(* CODESYS project Mini_Project.project

Project tree, tasks and I/O mapping:
  Device : CECC-LK, Festo AG & Co. KG, order no. 574418, version 3.5.4.0
    application Application
      libraries: Standard, * (System); Solution Center Library, 3.5.8.0 (Festo Didactic SE - Customer Solution Center); CAA CiA 405, 3.5.3.0 (CAA Technical Workgroup)
      task MainTask (cyclic, interval t#20ms, priority 20) calls PLC_PRG
      program PLC_PRG [ST]
      function block TCP_Conn [ST]
      function block RFID_Read [ST]
      function block SPLIT_String [ST]
      function formatMsg [ST]
    Onboard : CECC 14I/8O, Festo AG & Co. KG, version 3.4.5.5
        unmapped channels: Onboard Input, Onboard Output
      Digital Inputs
          unmapped channels: Onboard Input
      Digital Outputs
          unmapped channels: Onboard Output
    CANbus : CANbus, 3S - Smart Software Solutions GmbH, version 3.5.7.0
        settings: Baudrate = 1000
      CANopen_Manager : CANopen_Manager, 3S - Smart Software Solutions GmbH, version 3.5.10.0
          settings: ConfigVersion = 50659584
        BL20_GWBR_CANOPEN : BL20-GWBR-CANOPEN, TURCK, order no. 6827167, version Revision=16#00040017, FileVersion=4.23
            settings: General Options.Reset Node = FALSE; NODEIDSAVED = 2; SDO Timeout = 1000000; PDO_Autoconfig = TRUE; EXPERTSETTINGS = True; Emergency-General Parameters.Emergency COBID = 16#00000082; Settings.COBID = 16#00000202; Settings.Transmission Type = 16#FF; Settings.available PDO-Parameter.Inhibit Time available = FALSE; Settings.available PDO-Parameter.Event Timer available = FALSE; Settings.Inhibit Time = 0; Settings.Event Timer = 0; Generic COBID = '$NODEID+16#0200'; Settings.COBID = 16#00000302; Settings.Transmission Type = 16#FF; Settings.available PDO-Parameter.Inhibit Time available = FALSE; Settings.available PDO-Parameter.Event Timer available = FALSE; Settings.Inhibit Time = 0; Settings.Event Timer = 0; Generic COBID = '$NODEID+16#0300'; Settings.COBID = 16#00000182; Settings.Transmission Type = 16#FF; Settings.available PDO-Parameter.Inhibit Time available = TRUE; Settings.available PDO-Parameter.Event Timer available = TRUE; Settings.Inhibit Time = 0; Settings.Event Timer = 0; Generic COBID = '$NODEID+16#0180'; Settings.COBID = 16#00000282; Settings.Transmission Type = 16#FF; Settings.available PDO-Parameter.Inhibit Time available = TRUE; Settings.available PDO-Parameter.Event Timer available = TRUE; Settings.Inhibit Time = 0; Settings.Event Timer = 0; Generic COBID = '$NODEID+16#0280'; Heartbeat-Consuming1.Heartbeat-Time = 300 ms; WriteOutput8Bit : Generic_BL20_4DO.Index = 16#6200; WriteOutput8Bit : Generic_BL20_4DO.Subindex = 16#01; WriteOutput8Bit : Generic_BL20_4DO.ObjectLength = 8; WriteOutput8Bit : Generic_BL20_4DO_2.Index = 16#6200; WriteOutput8Bit : Generic_BL20_4DO_2.Subindex = 16#02;
              WriteOutput8Bit : Generic_BL20_4DO_2.ObjectLength = 8; WriteAnalogueOutput16 : Generic_BL20_2AO.Index = 16#6411; WriteAnalogueOutput16 : Generic_BL20_2AO.Subindex = 16#01; WriteAnalogueOutput16 : Generic_BL20_2AO.ObjectLength = 16; WriteAnalogueOutput16 : Generic_BL20_2AO.Index = 16#6411; WriteAnalogueOutput16 : Generic_BL20_2AO.Subindex = 16#02; WriteAnalogueOutput16 : Generic_BL20_2AO.ObjectLength = 16; ReadInput8Bit : Generic_BL20_4DI.Index = 16#6000; ReadInput8Bit : Generic_BL20_4DI.Subindex = 16#01; ReadInput8Bit : Generic_BL20_4DI.ObjectLength = 8; ReadAnalogueInput16Bit : Generic_BL20_4AI.Index = 16#6401; ReadAnalogueInput16Bit : Generic_BL20_4AI.Subindex = 16#01; ReadAnalogueInput16Bit : Generic_BL20_4AI.ObjectLength = 16; ReadAnalogueInput16Bit : Generic_BL20_4AI.Index = 16#6401; ReadAnalogueInput16Bit : Generic_BL20_4AI.Subindex = 16#02; ReadAnalogueInput16Bit : Generic_BL20_4AI.ObjectLength = 16; ReadAnalogueInput16Bit : Generic_BL20_4AI.Index = 16#6401; ReadAnalogueInput16Bit : Generic_BL20_4AI.Subindex = 16#03; ReadAnalogueInput16Bit : Generic_BL20_4AI.ObjectLength = 16; ReadAnalogueInput16Bit : Generic_BL20_4AI.Index = 16#6401; ReadAnalogueInput16Bit : Generic_BL20_4AI.Subindex = 16#04; ReadAnalogueInput16Bit : Generic_BL20_4AI.ObjectLength = 16; SDO List.Set Guardtime.Index = 16#100C; SDO List.Set Guardtime.Subindex = 16#00; SDO List.Set Guardtime.Value = 16#00000000; SDO List.Set Guardtime.Size = 16; SDO List.Set Guardtime.AbortIfError = FALSE; SDO List.Set Guardtime.JumpToLine = FALSE; SDO List.Set Guardtime.Line = 0; SDO List.Set Lifetime.Index = 16#100D; SDO List.Set Lifetime.Subindex = 16#00; SDO List.Set Lifetime.Value = 16#00000000; SDO List.Set Lifetime.Size = 8; SDO List.Set Lifetime.AbortIfError = FALSE; SDO List.Set Lifetime.JumpToLine = FALSE; SDO List.Set Lifetime.Line = 0; SDO List.Disable Emcy CobID.Index = 16#1014; SDO List.Disable Emcy CobID.Subindex = 16#00; SDO List.Disable Emcy CobID.Value = 16#80000082; SDO List.Disable Emcy CobID.Size = 32;
              SDO List.Disable Emcy CobID.AbortIfError = FALSE; SDO List.Disable Emcy CobID.JumpToLine = FALSE; SDO List.Disable Emcy CobID.Line = 0; SDO List.Set Emcy CobID.Index = 16#1014; SDO List.Set Emcy CobID.Subindex = 16#00; SDO List.Set Emcy CobID.Value = 16#00000082; SDO List.Set Emcy CobID.Size = 32; SDO List.Set Emcy CobID.AbortIfError = FALSE; SDO List.Set Emcy CobID.JumpToLine = FALSE; SDO List.Set Emcy CobID.Line = 0; SDO List.Set Heartbeat Consumer.Index = 16#1016; SDO List.Set Heartbeat Consumer.Subindex = 16#01; SDO List.Set Heartbeat Consumer.Value = 16#007F012C; SDO List.Set Heartbeat Consumer.Size = 32; SDO List.Set Heartbeat Consumer.AbortIfError = FALSE; SDO List.Set Heartbeat Consumer.JumpToLine = FALSE; SDO List.Set Heartbeat Consumer.Line = 0; SDO List.Set Heartbeat Producer.Index = 16#1017; SDO List.Set Heartbeat Producer.Subindex = 16#00; SDO List.Set Heartbeat Producer.Value = 16#00000000; SDO List.Set Heartbeat Producer.Size = 16; SDO List.Set Heartbeat Producer.AbortIfError = FALSE; SDO List.Set Heartbeat Producer.JumpToLine = FALSE; SDO List.Set Heartbeat Producer.Line = 0; SDO List.Disable PDO.Index = 16#1400; SDO List.Disable PDO.Subindex = 16#01; SDO List.Disable PDO.Value = 16#80000202; SDO List.Disable PDO.Size = 32; SDO List.Disable PDO.AbortIfError = FALSE; SDO List.Disable PDO.JumpToLine = FALSE; SDO List.Disable PDO.Line = 0; SDO List.Set transmission type.Index = 16#1400; SDO List.Set transmission type.Subindex = 16#02; SDO List.Set transmission type.Value = 16#FF; SDO List.Set transmission type.Size = 8; SDO List.Set transmission type.AbortIfError = FALSE; SDO List.Set transmission type.JumpToLine = FALSE; SDO List.Set transmission type.Line = 0; SDO List.Clear pdo mapping.Index = 16#1600; SDO List.Clear pdo mapping.Subindex = 16#00;
              SDO List.Clear pdo mapping.Value = 16#0; SDO List.Clear pdo mapping.Size = 8; SDO List.Clear pdo mapping.AbortIfError = FALSE; SDO List.Clear pdo mapping.JumpToLine = FALSE; SDO List.Clear pdo mapping.Line = 0; SDO List.Set Mapping.Index = 16#1600; SDO List.Set Mapping.Subindex = 16#01; SDO List.Set Mapping.Value = 16#62000108; SDO List.Set Mapping.Size = 32; SDO List.Set Mapping.AbortIfError = FALSE; SDO List.Set Mapping.JumpToLine = FALSE; SDO List.Set Mapping.Line = 0; SDO List.Set Mapping.Index = 16#1600; SDO List.Set Mapping.Subindex = 16#02; SDO List.Set Mapping.Value = 16#62000208; SDO List.Set Mapping.Size = 32; SDO List.Set Mapping.AbortIfError = FALSE; SDO List.Set Mapping.JumpToLine = FALSE; SDO List.Set Mapping.Line = 0; SDO List.Set number of mappings.Index = 16#1600; SDO List.Set number of mappings.Subindex = 16#00; SDO List.Set number of mappings.Value = 16#02; SDO List.Set number of mappings.Size = 8; SDO List.Set number of mappings.AbortIfError = FALSE; SDO List.Set number of mappings.JumpToLine = FALSE; SDO List.Set number of mappings.Line = 0; SDO List.Set and enable COB-ID.Index = 16#1400; SDO List.Set and enable COB-ID.Subindex = 16#01; SDO List.Set and enable COB-ID.Value = 16#00000202; SDO List.Set and enable COB-ID.Size = 32; SDO List.Set and enable COB-ID.AbortIfError = FALSE; SDO List.Set and enable COB-ID.JumpToLine = FALSE; SDO List.Set and enable COB-ID.Line = 0; SDO List.Disable PDO.Index = 16#1401; SDO List.Disable PDO.Subindex = 16#01; SDO List.Disable PDO.Value = 16#80000302; SDO List.Disable PDO.Size = 32; SDO List.Disable PDO.AbortIfError = FALSE; SDO List.Disable PDO.JumpToLine = FALSE; SDO List.Disable PDO.Line = 0;
              SDO List.Set transmission type.Index = 16#1401; SDO List.Set transmission type.Subindex = 16#02; SDO List.Set transmission type.Value = 16#FF; SDO List.Set transmission type.Size = 8; SDO List.Set transmission type.AbortIfError = FALSE; SDO List.Set transmission type.JumpToLine = FALSE; SDO List.Set transmission type.Line = 0; SDO List.Clear pdo mapping.Index = 16#1601; SDO List.Clear pdo mapping.Subindex = 16#00; SDO List.Clear pdo mapping.Value = 16#0; SDO List.Clear pdo mapping.Size = 8; SDO List.Clear pdo mapping.AbortIfError = FALSE; SDO List.Clear pdo mapping.JumpToLine = FALSE; SDO List.Clear pdo mapping.Line = 0; SDO List.Set Mapping.Index = 16#1601; SDO List.Set Mapping.Subindex = 16#01; SDO List.Set Mapping.Value = 16#64110110; SDO List.Set Mapping.Size = 32; SDO List.Set Mapping.AbortIfError = FALSE; SDO List.Set Mapping.JumpToLine = FALSE; SDO List.Set Mapping.Line = 0; SDO List.Set Mapping.Index = 16#1601; SDO List.Set Mapping.Subindex = 16#02; SDO List.Set Mapping.Value = 16#64110210; SDO List.Set Mapping.Size = 32; SDO List.Set Mapping.AbortIfError = FALSE; SDO List.Set Mapping.JumpToLine = FALSE; SDO List.Set Mapping.Line = 0; SDO List.Set number of mappings.Index = 16#1601; SDO List.Set number of mappings.Subindex = 16#00; SDO List.Set number of mappings.Value = 16#02; SDO List.Set number of mappings.Size = 8; SDO List.Set number of mappings.AbortIfError = FALSE; SDO List.Set number of mappings.JumpToLine = FALSE; SDO List.Set number of mappings.Line = 0; SDO List.Set and enable COB-ID.Index = 16#1401; SDO List.Set and enable COB-ID.Subindex = 16#01; SDO List.Set and enable COB-ID.Value = 16#00000302; SDO List.Set and enable COB-ID.Size = 32; SDO List.Set and enable COB-ID.AbortIfError = FALSE;
              SDO List.Set and enable COB-ID.JumpToLine = FALSE; SDO List.Set and enable COB-ID.Line = 0; SDO List.Disable PDO.Index = 16#1800; SDO List.Disable PDO.Subindex = 16#01; SDO List.Disable PDO.Value = 16#80000182; SDO List.Disable PDO.Size = 32; SDO List.Disable PDO.AbortIfError = FALSE; SDO List.Disable PDO.JumpToLine = FALSE; SDO List.Disable PDO.Line = 0; SDO List.Set transmission type.Index = 16#1800; SDO List.Set transmission type.Subindex = 16#02; SDO List.Set transmission type.Value = 16#FF; SDO List.Set transmission type.Size = 8; SDO List.Set transmission type.AbortIfError = FALSE; SDO List.Set transmission type.JumpToLine = FALSE; SDO List.Set transmission type.Line = 0; SDO List.Set inhibit time.Index = 16#1800; SDO List.Set inhibit time.Subindex = 16#03; SDO List.Set inhibit time.Value = 16#0000; SDO List.Set inhibit time.Size = 16; SDO List.Set inhibit time.AbortIfError = FALSE; SDO List.Set inhibit time.JumpToLine = FALSE; SDO List.Set inhibit time.Line = 0; SDO List.Set event time.Index = 16#1800; SDO List.Set event time.Subindex = 16#05; SDO List.Set event time.Value = 16#0000; SDO List.Set event time.Size = 16; SDO List.Set event time.AbortIfError = FALSE; SDO List.Set event time.JumpToLine = FALSE; SDO List.Set event time.Line = 0; SDO List.Clear pdo mapping.Index = 16#1A00; SDO List.Clear pdo mapping.Subindex = 16#00; SDO List.Clear pdo mapping.Value = 16#0; SDO List.Clear pdo mapping.Size = 8; SDO List.Clear pdo mapping.AbortIfError = FALSE; SDO List.Clear pdo mapping.JumpToLine = FALSE; SDO List.Clear pdo mapping.Line = 0; SDO List.Set Mapping.Index = 16#1A00; SDO List.Set Mapping.Subindex = 16#01; SDO List.Set Mapping.Value = 16#60000108;
              SDO List.Set Mapping.Size = 32; SDO List.Set Mapping.AbortIfError = FALSE; SDO List.Set Mapping.JumpToLine = FALSE; SDO List.Set Mapping.Line = 0; SDO List.Set number of mappings.Index = 16#1A00; SDO List.Set number of mappings.Subindex = 16#00; SDO List.Set number of mappings.Value = 16#01; SDO List.Set number of mappings.Size = 8; SDO List.Set number of mappings.AbortIfError = FALSE; SDO List.Set number of mappings.JumpToLine = FALSE; SDO List.Set number of mappings.Line = 0; SDO List.Set and enable COB-ID.Index = 16#1800; SDO List.Set and enable COB-ID.Subindex = 16#01; SDO List.Set and enable COB-ID.Value = 16#00000182; SDO List.Set and enable COB-ID.Size = 32; SDO List.Set and enable COB-ID.AbortIfError = FALSE; SDO List.Set and enable COB-ID.JumpToLine = FALSE; SDO List.Set and enable COB-ID.Line = 0; SDO List.Disable PDO.Index = 16#1801; SDO List.Disable PDO.Subindex = 16#01; SDO List.Disable PDO.Value = 16#80000282; SDO List.Disable PDO.Size = 32; SDO List.Disable PDO.AbortIfError = FALSE; SDO List.Disable PDO.JumpToLine = FALSE; SDO List.Disable PDO.Line = 0; SDO List.Set transmission type.Index = 16#1801; SDO List.Set transmission type.Subindex = 16#02; SDO List.Set transmission type.Value = 16#FF; SDO List.Set transmission type.Size = 8; SDO List.Set transmission type.AbortIfError = FALSE; SDO List.Set transmission type.JumpToLine = FALSE; SDO List.Set transmission type.Line = 0; SDO List.Set inhibit time.Index = 16#1801; SDO List.Set inhibit time.Subindex = 16#03; SDO List.Set inhibit time.Value = 16#0000; SDO List.Set inhibit time.Size = 16; SDO List.Set inhibit time.AbortIfError = FALSE; SDO List.Set inhibit time.JumpToLine = FALSE; SDO List.Set inhibit time.Line = 0; SDO List.Set event time.Index = 16#1801;
              SDO List.Set event time.Subindex = 16#05; SDO List.Set event time.Value = 16#0000; SDO List.Set event time.Size = 16; SDO List.Set event time.AbortIfError = FALSE; SDO List.Set event time.JumpToLine = FALSE; SDO List.Set event time.Line = 0; SDO List.Clear pdo mapping.Index = 16#1A01; SDO List.Clear pdo mapping.Subindex = 16#00; SDO List.Clear pdo mapping.Value = 16#0; SDO List.Clear pdo mapping.Size = 8; SDO List.Clear pdo mapping.AbortIfError = FALSE; SDO List.Clear pdo mapping.JumpToLine = FALSE; SDO List.Clear pdo mapping.Line = 0; SDO List.Set Mapping.Index = 16#1A01; SDO List.Set Mapping.Subindex = 16#01; SDO List.Set Mapping.Value = 16#64010110; SDO List.Set Mapping.Size = 32; SDO List.Set Mapping.AbortIfError = FALSE; SDO List.Set Mapping.JumpToLine = FALSE; SDO List.Set Mapping.Line = 0; SDO List.Set Mapping.Index = 16#1A01; SDO List.Set Mapping.Subindex = 16#02; SDO List.Set Mapping.Value = 16#64010210; SDO List.Set Mapping.Size = 32; SDO List.Set Mapping.AbortIfError = FALSE; SDO List.Set Mapping.JumpToLine = FALSE; SDO List.Set Mapping.Line = 0; SDO List.Set Mapping.Index = 16#1A01; SDO List.Set Mapping.Subindex = 16#03; SDO List.Set Mapping.Value = 16#64010310; SDO List.Set Mapping.Size = 32; SDO List.Set Mapping.AbortIfError = FALSE; SDO List.Set Mapping.JumpToLine = FALSE; SDO List.Set Mapping.Line = 0; SDO List.Set Mapping.Index = 16#1A01; SDO List.Set Mapping.Subindex = 16#04; SDO List.Set Mapping.Value = 16#64010410; SDO List.Set Mapping.Size = 32; SDO List.Set Mapping.AbortIfError = FALSE; SDO List.Set Mapping.JumpToLine = FALSE;
              SDO List.Set Mapping.Line = 0; SDO List.Set number of mappings.Index = 16#1A01; SDO List.Set number of mappings.Subindex = 16#00; SDO List.Set number of mappings.Value = 16#04; SDO List.Set number of mappings.Size = 8; SDO List.Set number of mappings.AbortIfError = FALSE; SDO List.Set number of mappings.JumpToLine = FALSE; SDO List.Set number of mappings.Line = 0; SDO List.Set and enable COB-ID.Index = 16#1801; SDO List.Set and enable COB-ID.Subindex = 16#01; SDO List.Set and enable COB-ID.Value = 16#00000282; SDO List.Set and enable COB-ID.Size = 32; SDO List.Set and enable COB-ID.AbortIfError = FALSE; SDO List.Set and enable COB-ID.JumpToLine = FALSE; SDO List.Set and enable COB-ID.Line = 0; ConfigVersion = 50659584
          Generic_BL20_2AO : Generic BL20-2AO, TURCK, order no. 0, version Revision=16#00040017, FileVersion=4.23
              settings: Number of Params = 2; WriteAnalogueOutput16 : Generic_BL20_2AO.Index = 16#6411; WriteAnalogueOutput16 : Generic_BL20_2AO.Subindex = 16#01; WriteAnalogueOutput16 : Generic_BL20_2AO.Startbit = 0; WriteAnalogueOutput16 : Generic_BL20_2AO.Endbit = 15; WriteAnalogueOutput16 : Generic_BL20_2AO.Index = 16#6411; WriteAnalogueOutput16 : Generic_BL20_2AO.Subindex = 16#02; WriteAnalogueOutput16 : Generic_BL20_2AO.Startbit = 0; WriteAnalogueOutput16 : Generic_BL20_2AO.Endbit = 15
              unmapped channels: WriteAnalogueOutput16 : Generic_BL20_2AO, WriteAnalogueOutput16 : Generic_BL20_2AO
          Generic_BL20_4AI : Generic BL20-4AI, TURCK, order no. 0, version Revision=16#00040017, FileVersion=4.23
              settings: Number of Params = 4; ReadAnalogueInput16Bit : Generic_BL20_4AI.Index = 16#6401; ReadAnalogueInput16Bit : Generic_BL20_4AI.Subindex = 16#01; ReadAnalogueInput16Bit : Generic_BL20_4AI.Startbit = 0; ReadAnalogueInput16Bit : Generic_BL20_4AI.Endbit = 15; ReadAnalogueInput16Bit : Generic_BL20_4AI.Index = 16#6401; ReadAnalogueInput16Bit : Generic_BL20_4AI.Subindex = 16#02; ReadAnalogueInput16Bit : Generic_BL20_4AI.Startbit = 0; ReadAnalogueInput16Bit : Generic_BL20_4AI.Endbit = 15; ReadAnalogueInput16Bit : Generic_BL20_4AI.Index = 16#6401; ReadAnalogueInput16Bit : Generic_BL20_4AI.Subindex = 16#03; ReadAnalogueInput16Bit : Generic_BL20_4AI.Startbit = 0; ReadAnalogueInput16Bit : Generic_BL20_4AI.Endbit = 15; ReadAnalogueInput16Bit : Generic_BL20_4AI.Index = 16#6401; ReadAnalogueInput16Bit : Generic_BL20_4AI.Subindex = 16#04; ReadAnalogueInput16Bit : Generic_BL20_4AI.Startbit = 0; ReadAnalogueInput16Bit : Generic_BL20_4AI.Endbit = 15
              unmapped channels: ReadAnalogueInput16Bit : Generic_BL20_4AI, ReadAnalogueInput16Bit : Generic_BL20_4AI, ReadAnalogueInput16Bit : Generic_BL20_4AI, ReadAnalogueInput16Bit : Generic_BL20_4AI
          Generic_BL20_4DO_3 : Generic BL20-4DO, TURCK, order no. 0, version Revision=16#00040017, FileVersion=4.23
              settings: Number of Params = 1; WriteOutput8Bit : Generic_BL20_4DO_2.Index = 16#6200; WriteOutput8Bit : Generic_BL20_4DO_2.Subindex = 16#02; WriteOutput8Bit : Generic_BL20_4DO_2.Startbit = 4; WriteOutput8Bit : Generic_BL20_4DO_2.Endbit = 7
              unmapped channels: WriteOutput8Bit : Generic_BL20_4DO_2
          Generic_BL20_4DO_2 : Generic BL20-4DO, TURCK, order no. 0, version Revision=16#00040017, FileVersion=4.23
              settings: Number of Params = 1; WriteOutput8Bit : Generic_BL20_4DO_2.Index = 16#6200; WriteOutput8Bit : Generic_BL20_4DO_2.Subindex = 16#02; WriteOutput8Bit : Generic_BL20_4DO_2.Startbit = 0; WriteOutput8Bit : Generic_BL20_4DO_2.Endbit = 3
              unmapped channels: WriteOutput8Bit : Generic_BL20_4DO_2
          Generic_BL20_4DO_1 : Generic BL20-4DO, TURCK, order no. 0, version Revision=16#00040017, FileVersion=4.23
              settings: Number of Params = 1; WriteOutput8Bit : Generic_BL20_4DO.Index = 16#6200; WriteOutput8Bit : Generic_BL20_4DO.Subindex = 16#01; WriteOutput8Bit : Generic_BL20_4DO.Startbit = 4; WriteOutput8Bit : Generic_BL20_4DO.Endbit = 7
              unmapped channels: WriteOutput8Bit : Generic_BL20_4DO
          Generic_BL20_4DO : Generic BL20-4DO, TURCK, order no. 0, version Revision=16#00040017, FileVersion=4.23
              settings: Number of Params = 1; WriteOutput8Bit : Generic_BL20_4DO.Index = 16#6200; WriteOutput8Bit : Generic_BL20_4DO.Subindex = 16#01; WriteOutput8Bit : Generic_BL20_4DO.Startbit = 0; WriteOutput8Bit : Generic_BL20_4DO.Endbit = 3
              unmapped channels: WriteOutput8Bit : Generic_BL20_4DO
          Generic_BL20_BR_PF : Generic BL20-BR/-PF, TURCK, order no. 0, version Revision=16#00040017, FileVersion=4.23
          Generic_BL20_4DI_1 : Generic BL20-4DI, TURCK, order no. 0, version Revision=16#00040017, FileVersion=4.23
              settings: Number of Params = 1; ReadInput8Bit : Generic_BL20_4DI.Index = 16#6000; ReadInput8Bit : Generic_BL20_4DI.Subindex = 16#01; ReadInput8Bit : Generic_BL20_4DI.Startbit = 4; ReadInput8Bit : Generic_BL20_4DI.Endbit = 7
              unmapped channels: ReadInput8Bit : Generic_BL20_4DI
          Generic_BL20_4DI : Generic BL20-4DI, TURCK, order no. 0, version Revision=16#00040017, FileVersion=4.23
              settings: Number of Params = 1; ReadInput8Bit : Generic_BL20_4DI.Index = 16#6000; ReadInput8Bit : Generic_BL20_4DI.Subindex = 16#01; ReadInput8Bit : Generic_BL20_4DI.Startbit = 0; ReadInput8Bit : Generic_BL20_4DI.Endbit = 3
              unmapped channels: ReadInput8Bit : Generic_BL20_4DI
        DTM425 : DTM425, ifm electronic gmbh, order no. DTM425, version Revision=16#00000000, FileVersion=8.2, File=DTM425.eds
            settings: NODEIDSAVED = 32; SDO Timeout = 1000000; PDO_Autoconfig = FALSE; EXPERTSETTINGS = True; Emergency-General Parameters.Emergency COBID = 16#000000A0; Heartbeat-Producer Time = 200; PDO 16#1400.COBID = 16#00000220; PDO 16#1401.COBID = 16#00000320; PDO 16#1402.COBID = 16#00000420; PDO 16#1403.COBID = 16#00000520; PDO 16#1800.COBID = 16#000001A0; PDO 16#1800.Event Timer = 0; PDO 16#1801.COBID = 16#000002A0; PDO 16#1801.Event Timer = 0; PDO 16#1802.COBID = 16#000003A0; PDO 16#1802.Event Timer = 0; PDO 16#1803.COBID = 16#000004A0; PDO 16#1803.Event Timer = 0; Write Data (mappable): Write Trigger.Subindex = 16#00; Write Data (mappable): Data_sub1.Subindex = 16#01; Write Data (mappable): Data_sub2.Subindex = 16#02; Write Data (mappable): Data_sub3.Subindex = 16#03; Device Status.Subindex = 16#00; Read Data (mappable): Data_sub1.Subindex = 16#01; Read Data (mappable): Data_sub2.Subindex = 16#02; Read Data (mappable): Data_sub3.Subindex = 16#03; SDO List.Disable Emcy CobID.Index = 16#1014; SDO List.Disable Emcy CobID.Subindex = 16#00; SDO List.Disable Emcy CobID.Value = 16#800000A0; SDO List.Disable Emcy CobID.Size = 32; SDO List.Disable Emcy CobID.AbortIfError = FALSE; SDO List.Disable Emcy CobID.JumpToLine = FALSE; SDO List.Disable Emcy CobID.Line = 0; SDO List.Set Emcy CobID.Index = 16#1014; SDO List.Set Emcy CobID.Subindex = 16#00; SDO List.Set Emcy CobID.Value = 16#000000A0; SDO List.Set Emcy CobID.Size = 32; SDO List.Set Emcy CobID.AbortIfError = FALSE; SDO List.Set Emcy CobID.JumpToLine = FALSE; SDO List.Set Emcy CobID.Line = 0;
              SDO List.Set Heartbeat Producer.Index = 16#1017; SDO List.Set Heartbeat Producer.Subindex = 16#00; SDO List.Set Heartbeat Producer.Value = 16#000000C8; SDO List.Set Heartbeat Producer.Size = 16; SDO List.Set Heartbeat Producer.AbortIfError = FALSE; SDO List.Set Heartbeat Producer.JumpToLine = FALSE; SDO List.Set Heartbeat Producer.Line = 0; SDO List.Disable PDO.Index = 16#1400; SDO List.Disable PDO.Subindex = 16#01; SDO List.Disable PDO.Value = 16#80000220; SDO List.Disable PDO.Size = 32; SDO List.Disable PDO.AbortIfError = FALSE; SDO List.Disable PDO.JumpToLine = FALSE; SDO List.Disable PDO.Line = 0; SDO List.Set transmission type.Index = 16#1400; SDO List.Set transmission type.Subindex = 16#02; SDO List.Set transmission type.Value = 16#FF; SDO List.Set transmission type.Size = 8; SDO List.Set transmission type.AbortIfError = FALSE; SDO List.Set transmission type.JumpToLine = FALSE; SDO List.Set transmission type.Line = 0; SDO List.Clear pdo mapping.Index = 16#1600; SDO List.Clear pdo mapping.Subindex = 16#00; SDO List.Clear pdo mapping.Value = 16#0; SDO List.Clear pdo mapping.Size = 8; SDO List.Clear pdo mapping.AbortIfError = FALSE; SDO List.Clear pdo mapping.JumpToLine = FALSE; SDO List.Clear pdo mapping.Line = 0; SDO List.Set Mapping.Index = 16#1600; SDO List.Set Mapping.Subindex = 16#01; SDO List.Set Mapping.Value = 16#230F0040; SDO List.Set Mapping.Size = 32; SDO List.Set Mapping.AbortIfError = FALSE; SDO List.Set Mapping.JumpToLine = FALSE; SDO List.Set Mapping.Line = 0; SDO List.Set number of mappings.Index = 16#1600; SDO List.Set number of mappings.Subindex = 16#00; SDO List.Set number of mappings.Value = 16#01; SDO List.Set number of mappings.Size = 8; SDO List.Set number of mappings.AbortIfError = FALSE;
              SDO List.Set number of mappings.JumpToLine = FALSE; SDO List.Set number of mappings.Line = 0; SDO List.Set and enable COB-ID.Index = 16#1400; SDO List.Set and enable COB-ID.Subindex = 16#01; SDO List.Set and enable COB-ID.Value = 16#00000220; SDO List.Set and enable COB-ID.Size = 32; SDO List.Set and enable COB-ID.AbortIfError = FALSE; SDO List.Set and enable COB-ID.JumpToLine = FALSE; SDO List.Set and enable COB-ID.Line = 0; SDO List.Disable PDO.Index = 16#1401; SDO List.Disable PDO.Subindex = 16#01; SDO List.Disable PDO.Value = 16#80000320; SDO List.Disable PDO.Size = 32; SDO List.Disable PDO.AbortIfError = FALSE; SDO List.Disable PDO.JumpToLine = FALSE; SDO List.Disable PDO.Line = 0; SDO List.Set transmission type.Index = 16#1401; SDO List.Set transmission type.Subindex = 16#02; SDO List.Set transmission type.Value = 16#FF; SDO List.Set transmission type.Size = 8; SDO List.Set transmission type.AbortIfError = FALSE; SDO List.Set transmission type.JumpToLine = FALSE; SDO List.Set transmission type.Line = 0; SDO List.Clear pdo mapping.Index = 16#1601; SDO List.Clear pdo mapping.Subindex = 16#00; SDO List.Clear pdo mapping.Value = 16#0; SDO List.Clear pdo mapping.Size = 8; SDO List.Clear pdo mapping.AbortIfError = FALSE; SDO List.Clear pdo mapping.JumpToLine = FALSE; SDO List.Clear pdo mapping.Line = 0; SDO List.Set Mapping.Index = 16#1601; SDO List.Set Mapping.Subindex = 16#01; SDO List.Set Mapping.Value = 16#230A0140; SDO List.Set Mapping.Size = 32; SDO List.Set Mapping.AbortIfError = FALSE; SDO List.Set Mapping.JumpToLine = FALSE; SDO List.Set Mapping.Line = 0; SDO List.Set number of mappings.Index = 16#1601; SDO List.Set number of mappings.Subindex = 16#00; SDO List.Set number of mappings.Value = 16#01;
              SDO List.Set number of mappings.Size = 8; SDO List.Set number of mappings.AbortIfError = FALSE; SDO List.Set number of mappings.JumpToLine = FALSE; SDO List.Set number of mappings.Line = 0; SDO List.Set and enable COB-ID.Index = 16#1401; SDO List.Set and enable COB-ID.Subindex = 16#01; SDO List.Set and enable COB-ID.Value = 16#00000320; SDO List.Set and enable COB-ID.Size = 32; SDO List.Set and enable COB-ID.AbortIfError = FALSE; SDO List.Set and enable COB-ID.JumpToLine = FALSE; SDO List.Set and enable COB-ID.Line = 0; SDO List.Disable PDO.Index = 16#1402; SDO List.Disable PDO.Subindex = 16#01; SDO List.Disable PDO.Value = 16#80000420; SDO List.Disable PDO.Size = 32; SDO List.Disable PDO.AbortIfError = FALSE; SDO List.Disable PDO.JumpToLine = FALSE; SDO List.Disable PDO.Line = 0; SDO List.Set transmission type.Index = 16#1402; SDO List.Set transmission type.Subindex = 16#02; SDO List.Set transmission type.Value = 16#FF; SDO List.Set transmission type.Size = 8; SDO List.Set transmission type.AbortIfError = FALSE; SDO List.Set transmission type.JumpToLine = FALSE; SDO List.Set transmission type.Line = 0; SDO List.Clear pdo mapping.Index = 16#1602; SDO List.Clear pdo mapping.Subindex = 16#00; SDO List.Clear pdo mapping.Value = 16#0; SDO List.Clear pdo mapping.Size = 8; SDO List.Clear pdo mapping.AbortIfError = FALSE; SDO List.Clear pdo mapping.JumpToLine = FALSE; SDO List.Clear pdo mapping.Line = 0; SDO List.Set Mapping.Index = 16#1602; SDO List.Set Mapping.Subindex = 16#01; SDO List.Set Mapping.Value = 16#230A0240; SDO List.Set Mapping.Size = 32; SDO List.Set Mapping.AbortIfError = FALSE; SDO List.Set Mapping.JumpToLine = FALSE; SDO List.Set Mapping.Line = 0; SDO List.Set number of mappings.Index = 16#1602;
              SDO List.Set number of mappings.Subindex = 16#00; SDO List.Set number of mappings.Value = 16#01; SDO List.Set number of mappings.Size = 8; SDO List.Set number of mappings.AbortIfError = FALSE; SDO List.Set number of mappings.JumpToLine = FALSE; SDO List.Set number of mappings.Line = 0; SDO List.Set and enable COB-ID.Index = 16#1402; SDO List.Set and enable COB-ID.Subindex = 16#01; SDO List.Set and enable COB-ID.Value = 16#00000420; SDO List.Set and enable COB-ID.Size = 32; SDO List.Set and enable COB-ID.AbortIfError = FALSE; SDO List.Set and enable COB-ID.JumpToLine = FALSE; SDO List.Set and enable COB-ID.Line = 0; SDO List.Disable PDO.Index = 16#1403; SDO List.Disable PDO.Subindex = 16#01; SDO List.Disable PDO.Value = 16#80000520; SDO List.Disable PDO.Size = 32; SDO List.Disable PDO.AbortIfError = FALSE; SDO List.Disable PDO.JumpToLine = FALSE; SDO List.Disable PDO.Line = 0; SDO List.Set transmission type.Index = 16#1403; SDO List.Set transmission type.Subindex = 16#02; SDO List.Set transmission type.Value = 16#FF; SDO List.Set transmission type.Size = 8; SDO List.Set transmission type.AbortIfError = FALSE; SDO List.Set transmission type.JumpToLine = FALSE; SDO List.Set transmission type.Line = 0; SDO List.Clear pdo mapping.Index = 16#1603; SDO List.Clear pdo mapping.Subindex = 16#00; SDO List.Clear pdo mapping.Value = 16#0; SDO List.Clear pdo mapping.Size = 8; SDO List.Clear pdo mapping.AbortIfError = FALSE; SDO List.Clear pdo mapping.JumpToLine = FALSE; SDO List.Clear pdo mapping.Line = 0; SDO List.Set Mapping.Index = 16#1603; SDO List.Set Mapping.Subindex = 16#01; SDO List.Set Mapping.Value = 16#230A0340; SDO List.Set Mapping.Size = 32; SDO List.Set Mapping.AbortIfError = FALSE; SDO List.Set Mapping.JumpToLine = FALSE;
              SDO List.Set Mapping.Line = 0; SDO List.Set number of mappings.Index = 16#1603; SDO List.Set number of mappings.Subindex = 16#00; SDO List.Set number of mappings.Value = 16#01; SDO List.Set number of mappings.Size = 8; SDO List.Set number of mappings.AbortIfError = FALSE; SDO List.Set number of mappings.JumpToLine = FALSE; SDO List.Set number of mappings.Line = 0; SDO List.Set and enable COB-ID.Index = 16#1403; SDO List.Set and enable COB-ID.Subindex = 16#01; SDO List.Set and enable COB-ID.Value = 16#00000520; SDO List.Set and enable COB-ID.Size = 32; SDO List.Set and enable COB-ID.AbortIfError = FALSE; SDO List.Set and enable COB-ID.JumpToLine = FALSE; SDO List.Set and enable COB-ID.Line = 0; SDO List.Disable PDO.Index = 16#1800; SDO List.Disable PDO.Subindex = 16#01; SDO List.Disable PDO.Value = 16#800001A0; SDO List.Disable PDO.Size = 32; SDO List.Disable PDO.AbortIfError = FALSE; SDO List.Disable PDO.JumpToLine = FALSE; SDO List.Disable PDO.Line = 0; SDO List.Set transmission type.Index = 16#1800; SDO List.Set transmission type.Subindex = 16#02; SDO List.Set transmission type.Value = 16#FF; SDO List.Set transmission type.Size = 8; SDO List.Set transmission type.AbortIfError = FALSE; SDO List.Set transmission type.JumpToLine = FALSE; SDO List.Set transmission type.Line = 0; SDO List.Set inhibit time.Index = 16#1800; SDO List.Set inhibit time.Subindex = 16#03; SDO List.Set inhibit time.Value = 16#00C8; SDO List.Set inhibit time.Size = 16; SDO List.Set inhibit time.AbortIfError = FALSE; SDO List.Set inhibit time.JumpToLine = FALSE; SDO List.Set inhibit time.Line = 0; SDO List.Clear pdo mapping.Index = 16#1A00; SDO List.Clear pdo mapping.Subindex = 16#00; SDO List.Clear pdo mapping.Value = 16#0; SDO List.Clear pdo mapping.Size = 8;
              SDO List.Clear pdo mapping.AbortIfError = FALSE; SDO List.Clear pdo mapping.JumpToLine = FALSE; SDO List.Clear pdo mapping.Line = 0; SDO List.Set Mapping.Index = 16#1A00; SDO List.Set Mapping.Subindex = 16#01; SDO List.Set Mapping.Value = 16#21500020; SDO List.Set Mapping.Size = 32; SDO List.Set Mapping.AbortIfError = FALSE; SDO List.Set Mapping.JumpToLine = FALSE; SDO List.Set Mapping.Line = 0; SDO List.Set number of mappings.Index = 16#1A00; SDO List.Set number of mappings.Subindex = 16#00; SDO List.Set number of mappings.Value = 16#01; SDO List.Set number of mappings.Size = 8; SDO List.Set number of mappings.AbortIfError = FALSE; SDO List.Set number of mappings.JumpToLine = FALSE; SDO List.Set number of mappings.Line = 0; SDO List.Set and enable COB-ID.Index = 16#1800; SDO List.Set and enable COB-ID.Subindex = 16#01; SDO List.Set and enable COB-ID.Value = 16#000001A0; SDO List.Set and enable COB-ID.Size = 32; SDO List.Set and enable COB-ID.AbortIfError = FALSE; SDO List.Set and enable COB-ID.JumpToLine = FALSE; SDO List.Set and enable COB-ID.Line = 0; SDO List.Disable PDO.Index = 16#1801; SDO List.Disable PDO.Subindex = 16#01; SDO List.Disable PDO.Value = 16#800002A0; SDO List.Disable PDO.Size = 32; SDO List.Disable PDO.AbortIfError = FALSE; SDO List.Disable PDO.JumpToLine = FALSE; SDO List.Disable PDO.Line = 0; SDO List.Set transmission type.Index = 16#1801; SDO List.Set transmission type.Subindex = 16#02; SDO List.Set transmission type.Value = 16#FF; SDO List.Set transmission type.Size = 8; SDO List.Set transmission type.AbortIfError = FALSE; SDO List.Set transmission type.JumpToLine = FALSE; SDO List.Set transmission type.Line = 0; SDO List.Set inhibit time.Index = 16#1801; SDO List.Set inhibit time.Subindex = 16#03;
              SDO List.Set inhibit time.Value = 16#00C8; SDO List.Set inhibit time.Size = 16; SDO List.Set inhibit time.AbortIfError = FALSE; SDO List.Set inhibit time.JumpToLine = FALSE; SDO List.Set inhibit time.Line = 0; SDO List.Clear pdo mapping.Index = 16#1A01; SDO List.Clear pdo mapping.Subindex = 16#00; SDO List.Clear pdo mapping.Value = 16#0; SDO List.Clear pdo mapping.Size = 8; SDO List.Clear pdo mapping.AbortIfError = FALSE; SDO List.Clear pdo mapping.JumpToLine = FALSE; SDO List.Clear pdo mapping.Line = 0; SDO List.Set Mapping.Index = 16#1A01; SDO List.Set Mapping.Subindex = 16#01; SDO List.Set Mapping.Value = 16#220A0140; SDO List.Set Mapping.Size = 32; SDO List.Set Mapping.AbortIfError = FALSE; SDO List.Set Mapping.JumpToLine = FALSE; SDO List.Set Mapping.Line = 0; SDO List.Set number of mappings.Index = 16#1A01; SDO List.Set number of mappings.Subindex = 16#00; SDO List.Set number of mappings.Value = 16#01; SDO List.Set number of mappings.Size = 8; SDO List.Set number of mappings.AbortIfError = FALSE; SDO List.Set number of mappings.JumpToLine = FALSE; SDO List.Set number of mappings.Line = 0; SDO List.Set and enable COB-ID.Index = 16#1801; SDO List.Set and enable COB-ID.Subindex = 16#01; SDO List.Set and enable COB-ID.Value = 16#000002A0; SDO List.Set and enable COB-ID.Size = 32; SDO List.Set and enable COB-ID.AbortIfError = FALSE; SDO List.Set and enable COB-ID.JumpToLine = FALSE; SDO List.Set and enable COB-ID.Line = 0; SDO List.Disable PDO.Index = 16#1802; SDO List.Disable PDO.Subindex = 16#01; SDO List.Disable PDO.Value = 16#800003A0; SDO List.Disable PDO.Size = 32; SDO List.Disable PDO.AbortIfError = FALSE; SDO List.Disable PDO.JumpToLine = FALSE; SDO List.Disable PDO.Line = 0;
              SDO List.Set transmission type.Index = 16#1802; SDO List.Set transmission type.Subindex = 16#02; SDO List.Set transmission type.Value = 16#FF; SDO List.Set transmission type.Size = 8; SDO List.Set transmission type.AbortIfError = FALSE; SDO List.Set transmission type.JumpToLine = FALSE; SDO List.Set transmission type.Line = 0; SDO List.Set inhibit time.Index = 16#1802; SDO List.Set inhibit time.Subindex = 16#03; SDO List.Set inhibit time.Value = 16#00C8; SDO List.Set inhibit time.Size = 16; SDO List.Set inhibit time.AbortIfError = FALSE; SDO List.Set inhibit time.JumpToLine = FALSE; SDO List.Set inhibit time.Line = 0; SDO List.Clear pdo mapping.Index = 16#1A02; SDO List.Clear pdo mapping.Subindex = 16#00; SDO List.Clear pdo mapping.Value = 16#0; SDO List.Clear pdo mapping.Size = 8; SDO List.Clear pdo mapping.AbortIfError = FALSE; SDO List.Clear pdo mapping.JumpToLine = FALSE; SDO List.Clear pdo mapping.Line = 0; SDO List.Set Mapping.Index = 16#1A02; SDO List.Set Mapping.Subindex = 16#01; SDO List.Set Mapping.Value = 16#220A0240; SDO List.Set Mapping.Size = 32; SDO List.Set Mapping.AbortIfError = FALSE; SDO List.Set Mapping.JumpToLine = FALSE; SDO List.Set Mapping.Line = 0; SDO List.Set number of mappings.Index = 16#1A02; SDO List.Set number of mappings.Subindex = 16#00; SDO List.Set number of mappings.Value = 16#01; SDO List.Set number of mappings.Size = 8; SDO List.Set number of mappings.AbortIfError = FALSE; SDO List.Set number of mappings.JumpToLine = FALSE; SDO List.Set number of mappings.Line = 0; SDO List.Set and enable COB-ID.Index = 16#1802; SDO List.Set and enable COB-ID.Subindex = 16#01; SDO List.Set and enable COB-ID.Value = 16#000003A0; SDO List.Set and enable COB-ID.Size = 32; SDO List.Set and enable COB-ID.AbortIfError = FALSE;
              SDO List.Set and enable COB-ID.JumpToLine = FALSE; SDO List.Set and enable COB-ID.Line = 0; SDO List.Disable PDO.Index = 16#1803; SDO List.Disable PDO.Subindex = 16#01; SDO List.Disable PDO.Value = 16#800004A0; SDO List.Disable PDO.Size = 32; SDO List.Disable PDO.AbortIfError = FALSE; SDO List.Disable PDO.JumpToLine = FALSE; SDO List.Disable PDO.Line = 0; SDO List.Set transmission type.Index = 16#1803; SDO List.Set transmission type.Subindex = 16#02; SDO List.Set transmission type.Value = 16#FF; SDO List.Set transmission type.Size = 8; SDO List.Set transmission type.AbortIfError = FALSE; SDO List.Set transmission type.JumpToLine = FALSE; SDO List.Set transmission type.Line = 0; SDO List.Set inhibit time.Index = 16#1803; SDO List.Set inhibit time.Subindex = 16#03; SDO List.Set inhibit time.Value = 16#00C8; SDO List.Set inhibit time.Size = 16; SDO List.Set inhibit time.AbortIfError = FALSE; SDO List.Set inhibit time.JumpToLine = FALSE; SDO List.Set inhibit time.Line = 0; SDO List.Clear pdo mapping.Index = 16#1A03; SDO List.Clear pdo mapping.Subindex = 16#00; SDO List.Clear pdo mapping.Value = 16#0; SDO List.Clear pdo mapping.Size = 8; SDO List.Clear pdo mapping.AbortIfError = FALSE; SDO List.Clear pdo mapping.JumpToLine = FALSE; SDO List.Clear pdo mapping.Line = 0; SDO List.Set Mapping.Index = 16#1A03; SDO List.Set Mapping.Subindex = 16#01; SDO List.Set Mapping.Value = 16#220A0340; SDO List.Set Mapping.Size = 32; SDO List.Set Mapping.AbortIfError = FALSE; SDO List.Set Mapping.JumpToLine = FALSE; SDO List.Set Mapping.Line = 0; SDO List.Set number of mappings.Index = 16#1A03; SDO List.Set number of mappings.Subindex = 16#00; SDO List.Set number of mappings.Value = 16#01;
              SDO List.Set number of mappings.Size = 8; SDO List.Set number of mappings.AbortIfError = FALSE; SDO List.Set number of mappings.JumpToLine = FALSE; SDO List.Set number of mappings.Line = 0; SDO List.Set and enable COB-ID.Index = 16#1803; SDO List.Set and enable COB-ID.Subindex = 16#01; SDO List.Set and enable COB-ID.Value = 16#000004A0; SDO List.Set and enable COB-ID.Size = 32; SDO List.Set and enable COB-ID.AbortIfError = FALSE; SDO List.Set and enable COB-ID.JumpToLine = FALSE; SDO List.Set and enable COB-ID.Line = 0; ConfigVersion = 50659584
            unmapped channels: Write Data (mappable): Write Trigger, Write Data (mappable): Data_sub1, Write Data (mappable): Data_sub2, Write Data (mappable): Data_sub3, Device Status, Read Data (mappable): Data_sub1, Read Data (mappable): Data_sub2, Read Data (mappable): Data_sub3
*)

// Device/Application/PLC_PRG
PROGRAM PLC_PRG
VAR
	/// Inputs ///
	IS_STOPPER_DOWN	AT %IX1.0	: BOOL;	// Stopper released
	CARR_AVAL		AT %IX1.1	: BOOL;	// Carrier available
	/// Outputs ///	
	STOPPER_DOWN	AT %QX1.0	: BOOL;	// Release stopper
	CONV_RIGHT		AT %QX0.4	: BOOL;	// Conveyor to the right
	// TCP //
	myTCP			: TCP_Conn;
	TCP_IP			: STRING := '172.20.40.42';
	TCP_PORT		: UINT := 1234;
	Tcp_msg			: STRING;
	TcpPlcActive	: BOOL;
	TcpOrderComp	: BOOL;
	// RFID //
	myRFID			: RFID_Read;
	rfidTag			: UINT;
	preRfidTag		: UINT;
	// Carrier VAR //
	numOfCarr		: ARRAY[0..5] OF INT := [0,0,0,0,0];
	carrID			: ARRAY[0..5] OF INT := [1,7,6,5,3]; // THIS is the carriers' acutual ID
	carrDone		: ARRAY[0..5] OF BOOL := [0,0,0,0,0];
	carrDelay		: INT;
	isCarrNew		: BOOL := TRUE;
	// Split String //
	SPLIT			: SPLIT_String;
	// Timer //
	Timer			: TON;
	// loop VAR //
	i				: INT;
	mainState		: INT;
END_VAR

CASE mainState OF 
	
	0:	// Trys to estabilish a connection and if connected reads the buffer 
		Tcp_msg := '';
		myTCP(TcpIp:=TCP_IP, TcpPort:=TCP_PORT, Tcp_Read:=TRUE);
		Tcp_msg := myTCP.Tcp_msgReceived;
		
		// Checks if the server sent the correct message/acknowlegement to initiate the procedure
		IF Tcp_msg = '0:0:0:0:0' THEN
			myTCP.Tcp_Read := FALSE;
			TcpPlcActive := TRUE;
			CONV_RIGHT := FALSE;
			TcpOrderComp := FALSE;
			mainState := 1;
		END_IF
		
	1:	// Sends a message to the server that the PLC is ready to receive further instructions
		Tcp_msg := '';
		Tcp_msg := formatMsg(bPlcActive:=TcpPlcActive, bCONV_RIGHT:=CONV_RIGHT, bIS_STOPPER_DOWN:=IS_STOPPER_DOWN, bOrderComp:=TcpOrderComp, iTag:=0);
		myTCP(msg:=Tcp_msg ,Tcp_Send:=TRUE);	// This msg bring the server into the ordering mode
		mainState := 2;
		
	2:	// The PLC trys to connect to the server and when connected reads the message with the instructions
		Tcp_msg := ''; 
		myTCP(Tcp_Read:=TRUE);
		Tcp_msg := myTCP.Tcp_msgReceived;
		
		// Checks that a proper instruction has been received
		IF Tcp_msg <> '0:0:0:0:0' THEN
			myTCP.Tcp_Read := FALSE;
			mainState := 3;
		ELSE
			mainState := 2;
		END_IF
		
	3:
		// Splits the received Tcp_msg at string_character(sAT:=':'). Ex. TcpMsg := '1:2:3:45:0';  
		SPLIT(str:=Tcp_msg, sAT:=':');
		FOR i:=0 TO (SPLIT.numOfSplits -1) DO
			numOfCarr[i] := BYTE_TO_INT(SPLIT.sSplit[i]);
		END_FOR
		CONV_RIGHT := TRUE;
		mainState := 4;
		
	4:	// Checks if the order from the server has been completed, if not then it continues to process the order
		IF carrDone[0] AND carrDone[1] AND carrDone[2] AND carrDone[3] AND carrDone[4] THEN	
			mainState := 6;
		ELSE
			mainState := 5;
		END_IF	
		
	5:	// Reads the RFID tags if a carrier is avaliable
		IF CARR_AVAL THEN
			myRFID();
			rfidTag := myRFID.rfid_tag;
			IF rfidTag <> preRfidTag AND isCarrNew THEN
				// Checks if the current carrier is one we want and if it is, then it gets checked of the list 
				FOR i:=0 TO (SPLIT.numOfSplits -1) DO
					IF carrID[i] = UINT_TO_INT(rfidTag) AND numOfCarr[i] > 0 THEN
						numOfCarr[i] := numOfCarr[i] -1;
						carrDelay := carrID[i];
					END_IF 
					IF numOfCarr[i] = 0 THEN
						carrDone[i] := TRUE;
					END_IF
				END_FOR
				preRfidTag := rfidTag;
				isCarrNew := FALSE;	
			// Checks if the timer needs to be applied 
			ELSIF isCarrNew = FALSE THEN
				Timer(IN:=TRUE, PT:=INT_TO_TIME(carrDelay *1000));
				// Checks if the wait time for the current carrier has passed
				IF Timer.Q THEN
					STOPPER_DOWN := TRUE;
					isCarrNew := TRUE;
					Timer(IN:=FALSE);
				END_IF
			END_IF
		END_IF
		// Checks if the stopper is down and if it is, then it get put back up again
		IF IS_STOPPER_DOWN THEN
			STOPPER_DOWN := FALSE;
			carrDelay := 0;
		END_IF
		mainState := 4;

	6:	// Sets the variable back into its initial stats, so its ready for the next order
		FOR i:=0 TO 4 DO
			carrDone[i] := 0;
		END_FOR
		// Stops the conveyor and sets the order as has been completed 
		CONV_RIGHT := FALSE;
		TcpOrderComp := TRUE;
		
		// Send back to the server that the order has been complete along with some other infomation
		Tcp_msg := '';
		Tcp_msg := formatMsg(bPlcActive:=TcpPlcActive, bCONV_RIGHT:=CONV_RIGHT, bIS_STOPPER_DOWN:=IS_STOPPER_DOWN, bOrderComp:=TcpOrderComp, iTag:=rfidTag);
		myTCP(msg:=Tcp_msg ,Tcp_Send:=TRUE);
		mainState := 0;
END_CASE

END_PROGRAM

// Device/Application/formatMsg
FUNCTION formatMsg : STRING
VAR_INPUT
	bPlcActive			: BOOL;
	bCONV_RIGHT			: BOOL;
	bIS_STOPPER_DOWN	: BOOL;
	bOrderComp			: BOOL;
	iTag				: UINT;
END_VAR
VAR
	TcpMsg				: STRING;
END_VAR


TcpMsg := CONCAT(INT_TO_STRING(BOOL_TO_INT(bPlcActive)), ':'); 
TcpMsg := CONCAT(TcpMsg, INT_TO_STRING(BOOL_TO_INT(bCONV_RIGHT)));
TcpMsg := CONCAT(TcpMsg, ':'); 
TcpMsg := CONCAT(TcpMsg, INT_TO_STRING(BOOL_TO_INT(bIS_STOPPER_DOWN)));
TcpMsg := CONCAT(TcpMsg, ':'); 
TcpMsg := CONCAT(TcpMsg, INT_TO_STRING(BOOL_TO_INT(bOrderComp)));
TcpMsg := CONCAT(TcpMsg, ':');  
TcpMsg := CONCAT(TcpMsg, UINT_TO_STRING(iTag));

formatMsg := TcpMsg;

END_FUNCTION

// Device/Application/TCP_Conn
FUNCTION_BLOCK TCP_Conn
VAR_INPUT
	TcpIp				: STRING;
	TcpPort				: UINT;
	Tcp_Send 			: BOOL;
	Tcp_Read			: BOOL;
	msg					: STRING;
END_VAR
VAR_OUTPUT
	Tcp_msgReceived		: STRING;
END_VAR
VAR
	// TCP_IP //
	TCP					: dc_ecp.TcpClientString;
	TcpData				: INT := 1024;
	TcpState			: INT;
	preTcp_msgReceived  : STRING;
	// TIMER //
	Timer				: TON;
END_VAR

CASE TcpState OF	
	0://Reset connection
		TCP.Reset();
		TcpState:=1;
	1: //Wait for ready
		IF TCP.xReady THEN
			TcpState := 2;
		END_IF
	2: //Connecting
		TCP.Connect(sIP:=TcpIp,uiPort:=TcpPort);
		TcpState := 3;
	3: //Check if its connected properly
		IF TCP.xConnected THEN
			TcpState := 4;
		ELSE 
			TcpState := 2; 
		END_IF
	4: //send data
		IF Tcp_Send THEN
			TCP.Send(sMessage:=msg);
			// Gives a small delay so that there is time to actually send the data 
			Timer(IN:=TRUE, PT:=INT_TO_TIME(100));
			IF Timer.Q THEN
				Tcp_SEND := FALSE;
				Timer(IN:=FALSE);
				TcpState := 0;
			END_IF
		ELSIF Tcp_Read THEN
			TCP.Receive();
			Tcp_msgReceived := TCP.sReceived;
			TcpState := 3;
			// Checks that we have received new data and is not just reading some old data again
			IF Tcp_msgReceived <> preTcp_msgReceived THEN
				Tcp_Read := FALSE;
				preTcp_msgReceived := Tcp_msgReceived;
				TcpState := 0;
			END_IF
		ELSE
			TcpState := 0;
		END_IF
END_CASE
TCP();

END_FUNCTION_BLOCK

// Device/Application/RFID_Read
FUNCTION_BLOCK RFID_Read
VAR_OUTPUT
	rfid_tag		: UINT;
END_VAR
VAR
	// RFID_VAR //
	RFIDReader		: dc_ecp.Dtm425;
	RFIDData		: dc_ecp.st_CPF_RfidData;
	RFIDState		: INT := 0;
	carrierID		: UINT := 0;
END_VAR

CASE RFIDState OF
	0:
		IF RFIDReader.xReady THEN
			RFIDState := 1;
		END_IF
	1:
		RFIDReader.Connect(usiNodeId:=32 , usiNetworkId:=0 , usiChannel:=1);
		RFIDState := 2;
	2:
		IF RFIDReader.xConnected THEN
			RFIDState := 3;
		ELSE
			RFIDState := 1;
		END_IF
	3:
		RFIDReader.ReadTag(uiStartAddress := 0, uiDataLength := SIZEOF(RFIDData), ADR(RFIDData));	
		RFIDState := 4;
	4:
		carrierID := dc_ecp.SwapWORD(RFIDData.uiCarrierID);
		rfid_tag := carrierID;	
		RFIDState := 3;	
END_CASE
RFIDReader();

END_FUNCTION_BLOCK

// Device/Application/SPLIT_String
FUNCTION_BLOCK SPLIT_String
VAR_INPUT
	str				: STRING;
	sAT				: STRING;
END_VAR
VAR_OUTPUT
	sSplit			: STRING[50];
	numOfSplits		: INT;
END_VAR
VAR
	split			: BOOL := TRUE;
	charPos			: INT;
	strArray		: STRING[50];
END_VAR

// Splits a string with five entries all seperated be a ":" i.e TcpMsg := '1:2:3:45:0'; //
numOfSplits := 0;
WHILE split DO
	charPos := FIND(str, sAT);
	IF charPos = 0 THEN
		split := FALSE;
		charPos := LEN(str);
	END_IF
	strArray[numOfSplits] := STRING_TO_BYTE(LEFT(str, charPos));
	str := DELETE(str, LEN:=charPos, POS:=1);
	numOfSplits := numOfSplits +1;
END_WHILE

sSplit := strArray;

END_FUNCTION_BLOCK
